// TIA Portal V20 export
TYPE "LKinCtrl_typeSPTPDynamics"
   STRUCT
      velocityFactor : LReal := -1.0;   // Factor for the velocity of axis movements in relation to the respective maximum velocity of the axes. Permitted value range: -1.0 < Factor ≤ 1.0
      accelerationFactor : LReal := -1.0;   // Factor for the acceleration of axis movements in relation to the respective maximum acceleration of the axis. Permitted value range: -1.0 < Factor ≤ 1.0
      decelerationFactor : LReal := -1.0;   // Factor for the deceleration of the axis movements in relation to the respective maximum deceleration of the axis. Permitted value range: -1.0 < Factor ≤ 1.0
      jerkFactor : LReal := -1.0;   // Factor for the jerk of axis movements in relation to the respective maximum jerk of the axis. Permitted value range: -1.0 <Factor ≤ 0.0 and 0.1 < Factor ≤ 0.9
   END_STRUCT;
END_TYPE
